// TIA Portal V16 export
// export: Created 2021-03-04T22:04:04.7895578Z, ExportSetting WithDefaults, DisplayName Totally Integrated Automation Portal, DisplayVersion V16, DisplayName TIA Portal Version Control Interface, DisplayVersion V16, DisplayName TIA Portal Openness, DisplayVersion V16, DisplayName SINAMICS Startdrive Advanced, DisplayVersion V16, DisplayName SINAMICS Startdrive G130, G150, S120, S150, SINAMICS MV, S210, DisplayVersion V16, DisplayName SINAMICS Startdrive G110M, G120, G120C, G120D, G120P, DisplayVersion V16, DisplayName STEP 7 Professional, DisplayVersion V16, DisplayName STEP 7 Safety, DisplayVersion V16, DisplayName WinCC Professional, DisplayVersion V16
VAR_GLOBAL   // PLC tag table "GLOBAL_CONSTANTS"
END_VAR
VAR_GLOBAL CONSTANT   // user constants
   NUM_AI_RACK : UInt := 1;   // Number of physical analog input points used per rack.
   NUM_DQ_RACK : UInt := 4;   // Number of physical digital output points used per rack.
   NUM_DQ_ROOM : UInt := 9;   // Number of physical digital output points used per room.
   MAX_DQ_PER_ROOM : UInt := 40;   // Max number of physical digital output points per room-based IO module. This needs to equal (NUM_DQ_ROOM + NUM_DQ_RACK*MAX_RACKS_PER_ROOM + EXTRA_DQ_PER_ROOM).
   MAX_VFDS : UInt := 6;   // Total number of VFDs configured in the HW config. This needs to equal MAX_ROOMS * MAX_RACKS_PER_ROOM.
   MAX_ROOMS : UInt := 1;   // Maximum possible number of rooms controlled by a given PLC
   MAX_RACKS_PER_ROOM : UInt := 6;   // Maximum possible number of racks per room
   NUM_AI_ROOM : UInt := 13;   // Number of physical analog input points used per room.
   EXTRA_DQ_PER_ROOM : UInt := 7;   // Number of unused physical digital output points per room-based IO module.
   EXTRA_AI_PER_ROOM : UInt := 1;   // Number of unused physical analog input points per room-based IO module.
   MAX_AI_PER_ROOM : UInt := 20;   // Max number of physical analog input points per room-based IO module. This needs to equal (NUM_AI_ROOM + NUM_AI_RACK*MAX_RACKS_PER_ROOM + EXTRA_AI_PER_ROOM).
END_VAR
